(* CODESYS project PLCTEST.project
   Title: PLCTEST
   Author: Peter
   Version: 0.0.0.33

Project tree, tasks and I/O mapping:
  MyController_1 : TM241CEC24T/U, Schneider Electric, order no. TM241CEC24T/U, version 4.0.6.18
    application Application
      libraries: HMISCU PTOPWM, 2.0.1.4 (Schneider Electric); SM3_Basic, 3.5.3.83 (3S - Smart Software Solutions GmbH); PLCCommunication, 1.0.3.3 (Schneider Electric)
      task MAST (cyclic, interval 2 ms, priority 15, watchdog 100 ms x 1) calls POU_TEST, Modbus_pou
      task tProfibus (cyclic, interval T#100ms, priority 30) calls nothing
      program POU_TEST [ST]
      global variables GVL
      program POU [CFC]
      visualisation GUITest
      Symbols
      program Modbus_pou [ST]
    DI : Digital Inputs, Schneider Electric, version 4.0.6.18
        input  iwDI_IW0 : WORD  // IW0
        input  ibDI_IB1 : BYTE  // IB1
    DQ : Digital Outputs, Schneider Electric, version 4.0.6.18
        output Application.POU_TEST.plc_q7_en : BOOL  // QW0.Q7
        output Application.POU_TEST.plc_q8_en : BOOL  // QW0.Q8
        output Application.POU_TEST.plc_q9_en : BOOL  // QW0.Q9
        unmapped channels: QW0, QB1
    Counters : Counters, Schneider Electric, version 4.0.6.18
    Pulse_Generators : Pulse Generators, Schneider Electric, version 4.0.6.18
    Cartridge_1 : Cartridge, Schneider Electric, version 4.0.6.18
    IO_Bus : IO bus - TM3, Schneider Electric, version 4.0.6.18
      Module_1 : TM3SAF5R/G, Schneider Electric, order no. TM3SAF5R/G, version 1.0.1.12
          output Application.POU_TEST.tm_saf_en : BOOL  // QB0.Enable
          unmapped channels: IW0, QB0
      Module_2 : TM3AQ4/G, Schneider Electric, order no. TM3AQ4/G, version 1.0.0.12
          settings: KPI Configuration.KPI Configuration[1] = 17; KPI Configuration.KPI Configuration[6] = 240; KPI Configuration.KPI Configuration[7] = 216; KPI Configuration.KPI Configuration[14] = 16; KPI Configuration.KPI Configuration[15] = 39
          output qiModule_2_QW0 : INT  // QW0
          output Application.POU_TEST.tm_a_val : INT  // QW1
          output qiModule_2_QW2 : INT  // QW2
          output qiModule_2_QW3 : INT  // QW3
          input  ibModule_2_IBStatusQW0 : BYTE  // IBStatusQW0
          input  ibModule_2_IBStatusQW1 : BYTE  // IBStatusQW1
          input  ibModule_2_IBStatusQW2 : BYTE  // IBStatusQW2
          input  ibModule_2_IBStatusQW3 : BYTE  // IBStatusQW3
    COM_Bus : COM bus, Schneider Electric, version 4.0.6.18
    Ethernet_1 : Ethernet Network, Schneider Electric, version 4.0.6.18
        settings: IPAddress = [192, 168, 1, 180]; SubnetMask = [255, 255, 255, 0]; WebServer = TRUE; FTP Server = TRUE; SoMachine Protocol = TRUE; Modbus Server = TRUE; NetManage Protocol = TRUE; SNMP protocol = TRUE; Enable Routing = FALSE; WebVisu protocol = TRUE; DHCP Server Active = TRUE
    Serial_Line_1 : Serial line, Schneider Electric, version 4.0.6.18
      Modbus_IOScanner : Modbus IOScanner, Schneider Electric, version 3.5.3.8
        Generic_Modbus_Slave : Generic Modbus Slave, Schneider Electric, version 3.5.3.9
            settings: 16#0000 (=0).Function Code = 5; 16#0000 (=0).Write Offset = 0; 16#0000 (=0).Write Length = 1; 16#0000 (=0).Init Value = 1; Channel 1.Function Code = 23; Channel 1.Read Offset = 16#0000; Channel 1.Read Length = 1; Channel 1.Write Offset = 16#0000; Channel 1.Write Length = 1; Channel 1.Cycle Time = 100
            unmapped channels: Channel 1, Channel 1, Channel 1
    Serial_Line_2 : Serial line, Schneider Electric, version 4.0.6.18
      Modbus_IOScanner_1 : Modbus IOScanner, Schneider Electric, version 3.5.3.8
        Generic_Modbus_Slave_1 : Generic Modbus Slave, Schneider Electric, version 3.5.3.9
    CAN_1 : CANopen bus, Schneider Electric, version 4.0.6.18
        settings: BlockFDTSDO = FALSE
  FdtConnections : FDT Connections, Schneider Electric, version 1.0.0.2
    Modbus_Serial_Line_Manager : Modbus Serial Line Manager, Schneider Electric, version 2.2.5
      Lexium_32_C : Lexium 32 C Advanced Settings, Schneider Electric, version 1.18.00.07
  text list GlobalTextList
*)

// MyController_1/Application/GVL
VAR_GLOBAL
END_VAR

// MyController_1/Application/POU_TEST
PROGRAM POU_TEST
VAR
	tm_saf_en: BOOL;
	plc_q7_en: BOOL;
	plc_q8_en: BOOL;
	plc_q9_en: BOOL;
	tm_a_val: INT;
	dir: BOOL;
	timer: TON;
	enable: BOOL;
	gain: INT := 1;
	tid: TIME := T#1s;
END_VAR

IF enable THEN
	timer.PT := tid;
	timer.IN := TRUE;

	IF timer.Q THEN
		IF tm_a_val = 100 * gain THEN
			tm_a_val := -100 * gain;
		ELSE
			tm_a_val := 100 * gain;
		END_IF
		timer.IN := FALSE;
	END_IF
ELSE
	tm_a_val := 0;
END_IF


timer();

END_PROGRAM

// MyController_1/Application/Modbus_pou
PROGRAM Modbus_pou
VAR
	

(**********************)     (*** ADDM Variables ***)     (**********************)     
// ADDM Function Block for formatting the address of the ATV12 Modbus Slave     
	ADDM_MODBUS_ATV12           : ADDM;    
// ADDRESS structure for the address of the ATV12 Modbus Slave     
	v_addressModbusAtv12        : ADDRESS;     
// "Done" result of the Address conversion     
	v_xAddressDone              : BOOL :=   FALSE;    
// "Error" result of the Address conversion     
	v_xAddressError             : BOOL :=   FALSE;    
// Result of the Address conversion: OK if "Done" without any "Error"     
	v_xAddressIsOK              : BOOL :=   FALSE;
	
	linkNumber : LinkNumber;
	
	
	
END_VAR


//v_addressModbusAtv12.Link := linkNumber;
ADDM_MODBUS_ATV12(     
	AddrTable := v_addressModbusAtv12,  
// IN/OUT - Resulting ADDRESS structure     
		Execute   := TRUE,     
		
// IN     - Rising Edge signal that triggers    
	Addr      :=   '1.1');
    v_xAddressDone := ADDM_MODBUS_ATV12.Done;

END_PROGRAM

// MyController_1/Application/POU
PROGRAM POU
VAR
	MC_Power_LXM_0: MC_Power_LXM;
	MC_ReadActualVelocity_LXM_0: MC_ReadActualVelocity_LXM;
	MC_MoveVelocity_LXM_0: MC_MoveVelocity_LXM;
	MC_Reset_LXM_0: MC_Reset_LXM;
	MC_ReadStatus_LXM_0 : MC_ReadStatus_LXM;
	xPower: BOOL;
	xReset: BOOL;
	MC_Stop_LXM_0: MC_Stop_LXM;
	xStop: BOOL;
	xMove: BOOL;
END_VAR

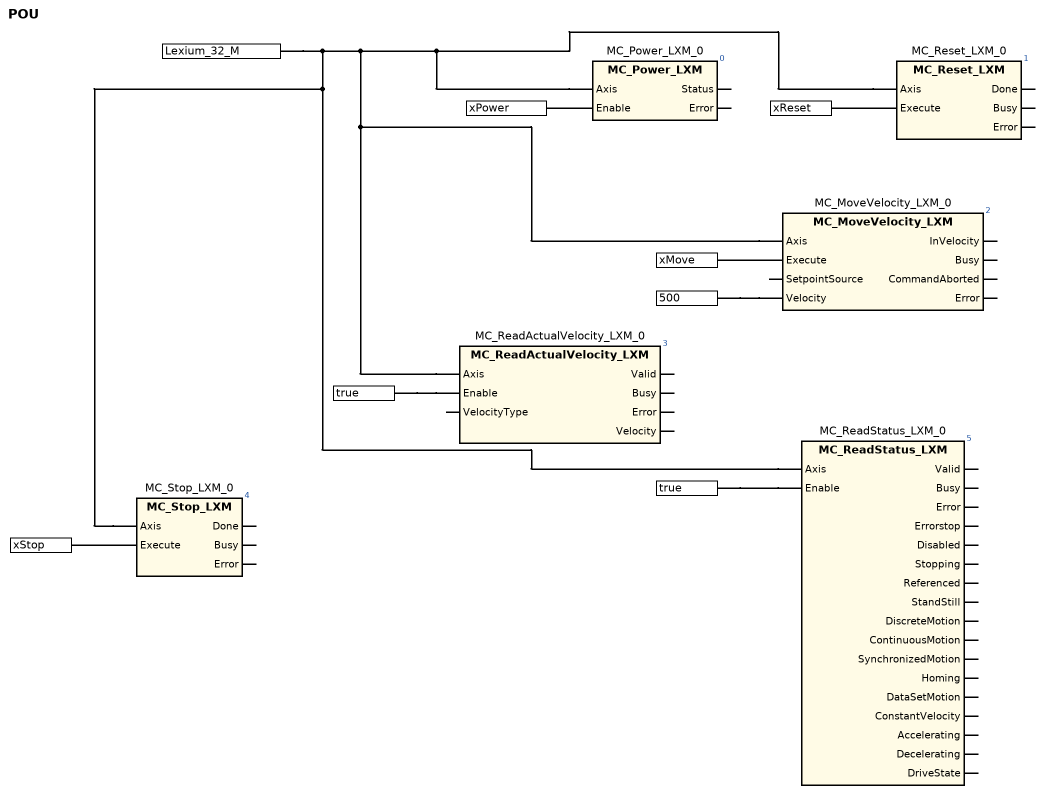
MC_Power_LXM_0(Axis := Lexium_32_M, Enable := xPower); // MC_Power_LXM
MC_Reset_LXM_0(Axis := Lexium_32_M, Execute := xReset); // MC_Reset_LXM
MC_MoveVelocity_LXM_0(Axis := Lexium_32_M, Execute := xMove, Velocity := 500); // MC_MoveVelocity_LXM
MC_ReadActualVelocity_LXM_0(Axis := Lexium_32_M, Enable := true); // MC_ReadActualVelocity_LXM
MC_Stop_LXM_0(Axis := Lexium_32_M, Execute := xStop); // MC_Stop_LXM
MC_ReadStatus_LXM_0(Axis := Lexium_32_M, Enable := true); // MC_ReadStatus_LXM

END_PROGRAM

// MyController_1/Application/GUITest
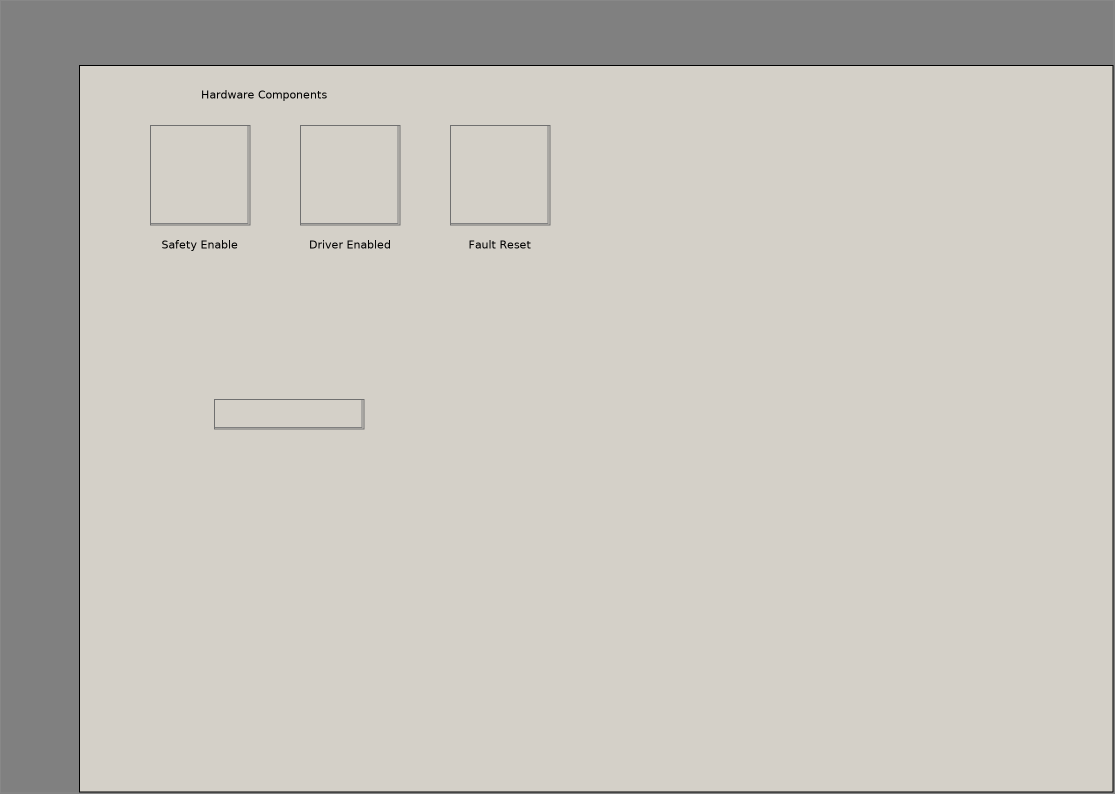
VISUALIZATION GUITest  // 1115x794
    Rectangle (79,65 1034x727)
    Button (150,125 100x100), colour toggle: POU_TEST.tm_saf_en
        toggle POU_TEST.tm_saf_en
    Button (300,125 100x100), colour toggle: POU_TEST.plc_q7_en
        toggle POU_TEST.plc_q7_en
    Label (150,230 100x30), "Safety Enable"
    Label (300,230 100x30), "Driver Enabled"
    Label (189,80 150x30), "Hardware Components"
    Button (450,125 100x100), colour toggle: POU_TEST.plc_q8_en
        toggle POU_TEST.plc_q8_en
    Label (450,230 100x30), "Fault Reset"
    Label (150,450 100x30)
    Label (150,600 100x30)
    Label (950,620 150x30)
    Button (214,399 150x30), colour toggle: POU_TEST.plc_q9_en
        toggle POU_TEST.plc_q9_en
END_VISUALIZATION
